FUNCTION_BLOCK FB_MotionShareData IMPLEMENTS I_MotionShareData
VAR_INPUT
END_VAR
VAR_OUTPUT
END_VAR
VAR
    (* Hardware *)
   // NC Forward Limit Switch: TRUE if ok to move
    bLimitForwardEnable AT %I*: BOOL;
    // NC Backward Limit Switch: TRUE if ok to move
    bLimitBackwardEnable AT %I*: BOOL;
    // NO Home Switch: TRUE if at home
    bHome AT %I*: BOOL;
END_VAR

{warning 'Add property implementation'}
(* Reads get this status from Interlock block*)
PROPERTY AllBackwardEnabled : BOOL
GET
END_GET
SET
END_SET
END_PROPERTY

{warning 'Add property implementation'}
(* Reads get this status from Interlock block*)
PROPERTY AllEnabled : BOOL
GET
END_GET
SET
END_SET
END_PROPERTY

{warning 'Add property implementation'}
(* Reads get this status from Interlock block*)
PROPERTY AllForwardEnabled : BOOL
GET
END_GET
SET
END_SET
END_PROPERTY

{warning 'Add property implementation'}
PROPERTY AxisError : BOOL
GET
END_GET
SET
END_SET
END_PROPERTY

{warning 'Add property implementation'}
PROPERTY AxisErrorID : UDINT
GET
END_GET
SET
END_SET
END_PROPERTY

{warning 'Add property implementation'}
PROPERTY AxisState : MC_AxisStates
GET
END_GET
SET
END_SET
END_PROPERTY

{warning 'Add property implementation'}
PROPERTY BrakeError : BOOL
GET
END_GET
END_PROPERTY

{warning 'Add property implementation'}
PROPERTY DriveEnable : BOOL
GET
END_GET
SET
END_SET
END_PROPERTY

{warning 'Add property implementation'}
PROPERTY ExecHome : BOOL
GET
END_GET
SET
END_SET
END_PROPERTY

{warning 'Add property implementation'}
PROPERTY ExecMove : BOOL
GET
END_GET
SET
END_SET
END_PROPERTY

{warning 'Add property implementation'}
PROPERTY GlobalReset : BOOL
GET
END_GET
SET
END_SET
END_PROPERTY

{warning 'Add property implementation'}
PROPERTY HomeBusy : BOOL
GET
END_GET
SET
END_SET
END_PROPERTY

{warning 'Add property implementation'}
PROPERTY InterlockOk : BOOL
GET
END_GET
END_PROPERTY

{warning 'Add property implementation'}
PROPERTY LimBackward : BOOL
GET
END_GET
END_PROPERTY

{warning 'Add property implementation'}
PROPERTY LimBwdEnable : BOOL
GET
END_GET
SET
END_SET
END_PROPERTY

{warning 'Add property implementation'}
PROPERTY LimForward : BOOL
GET
END_GET
END_PROPERTY

{warning 'Add property implementation'}
PROPERTY LimFwdEnable : BOOL
GET
END_GET
SET
END_SET
END_PROPERTY

{warning 'Add property implementation'}
PROPERTY LimHome : BOOL
GET
END_GET
SET
END_SET
END_PROPERTY

{warning 'Add property implementation'}
PROPERTY MoveBusy : BOOL
GET
END_GET
SET
END_SET
END_PROPERTY

{warning 'Add property implementation'}
PROPERTY NegativeDirection : BOOL
GET
END_GET
SET
END_SET
END_PROPERTY

{warning 'Add property implementation'}
PROPERTY NewMoveReq : BOOL
GET
END_GET
SET
END_SET
END_PROPERTY

{warning 'Add property implementation'}
PROPERTY PositiveDirection : BOOL
GET
END_GET
SET
END_SET
END_PROPERTY

{warning 'Add property implementation'}
PROPERTY ResetDone : BOOL
GET
END_GET
SET
END_SET
END_PROPERTY

{warning 'Add property implementation'}
PROPERTY RestoreDone : BOOL
GET
END_GET
SET
END_SET
END_PROPERTY

{warning 'Add property implementation'}
PROPERTY SavedPosition : LREAL
GET
END_GET
SET
END_SET
END_PROPERTY

{warning 'Add property implementation'}
PROPERTY ServoMode : BOOL
GET
END_GET
SET
END_SET
END_PROPERTY

END_FUNCTION_BLOCK

(* stored: Version 1.1.0.1
   POU FB_MotionShareData: Id {1501870c-92ad-4102-b185-4e7588eab041}, SpecialFunc None
   Property AllBackwardEnabled: Id {588933f9-668c-428c-b209-3fec4ae435c4}
   Get Get: Id {6ea50c3d-e5d3-4a80-b52c-1c3edbe55417}
   Set Set: Id {6c150d12-d1b5-4f4d-b7b7-ed56a08b0c53}
   Property AllEnabled: Id {531ae454-b142-4ec8-a6a5-51ea163f0f3b}
   Get Get: Id {35565f8a-1ea5-48a2-b92f-f1487a4c2726}
   Set Set: Id {b6605eb0-8b6e-487f-9c94-198c166233d5}
   Property AllForwardEnabled: Id {dd99efed-b46c-49c9-8796-4833ffe44a8e}
   Get Get: Id {21a84f27-171b-49b3-9d0a-8f77c1dec2a2}
   Set Set: Id {52d9b336-5323-4b37-acf3-5ca81300271c}
   Property AxisError: Id {98115272-2230-4767-b0dd-a49f097a3ce0}
   Get Get: Id {e08aea0a-ecc7-413f-a52a-c1e096c0cdf2}
   Set Set: Id {ef9e3f03-340b-499d-8070-7455ab14d8b6}
   Property AxisErrorID: Id {82dfdcd5-32b1-4e94-8a55-340757d1a7f1}
   Get Get: Id {6103d67a-1983-4236-bf4f-2f78135d229b}
   Set Set: Id {5a212e82-8ce0-4c2f-902b-ae2bc37a5cb5}
   Property AxisState: Id {cbea8871-01a0-4b37-8843-c349d6db3a77}
   Get Get: Id {b9c71475-3794-4e3a-82d7-abf6846e39f1}
   Set Set: Id {d1f98ffb-2b3d-4782-963e-39e553811b18}
   Property BrakeError: Id {b9794475-3295-45c0-b288-6d33ca0368ce}
   Get Get: Id {62ef9884-1fbf-41d5-b658-cf66ef51b265}
   Property DriveEnable: Id {dfcd0fcb-dffb-406f-b1e7-6950fa15a46c}
   Get Get: Id {db2324e9-bd6a-4fe7-9ec3-8b18495597ce}
   Set Set: Id {c3e3b36f-d36f-4e02-a404-47899aa59852}
   Property ExecHome: Id {89b20d8a-af4d-4bf3-9b64-5b77a7d8352f}
   Get Get: Id {16b7fe84-b047-4a79-80cb-896a9cb18e43}
   Set Set: Id {b29dda69-3987-4144-b0ee-0ba647ec0cf2}
   Property ExecMove: Id {91e258d6-97f4-47e1-9706-a43bc5f21419}
   Get Get: Id {a71b7848-fe39-473b-ac1e-c9df03bba908}
   Set Set: Id {3910c9d7-0829-4fb0-85f0-08cca942bd4f}
   Property GlobalReset: Id {323a9cf3-a3b0-42dc-b822-f29eb0e15c95}
   Get Get: Id {e42e6468-57d6-4eab-9213-e7eb1faa8826}
   Set Set: Id {fc8bced8-d33a-40ea-b8e4-9002dc5933ad}
   Property HomeBusy: Id {47aec562-24c8-4255-ab98-d9218f40240f}
   Get Get: Id {0cf0c789-b3ef-4e34-a21a-ea19e348b455}
   Set Set: Id {262b3e6f-6e52-4040-b215-b800b0158e51}
   Property InterlockOk: Id {3a9856fd-4650-49a0-b2fe-c96cc21117fa}
   Get Get: Id {fe0d79c1-f8f4-42e6-9406-9ec361dab8da}
   Property LimBackward: Id {38e5cd98-f346-4d1d-b128-21f2a07d0784}
   Get Get: Id {28999aa8-3674-4ecb-837f-ebb6de69864a}
   Property LimBwdEnable: Id {f6c9be89-9e8e-43ba-b22f-6910f8c266ad}
   Get Get: Id {21396ad7-f3b5-49e2-a94a-0f2ee23cefba}
   Set Set: Id {b68a63ad-3fa3-4f13-87d4-08acdd5974b5}
   Property LimForward: Id {58508ad6-a56e-4f16-90a2-2e7368217430}
   Get Get: Id {6df200ef-9186-43a2-ab57-1b46b7ba3ed7}
   Property LimFwdEnable: Id {7abd22ed-a794-45d0-86da-9a21cd25e8a9}
   Get Get: Id {ccece1fc-0a1c-4316-bb2a-391f9e29b850}
   Set Set: Id {58a697a9-c461-4dde-955a-f98b0dcfea88}
   Property LimHome: Id {4024a463-7a7f-421e-a252-cf6b7e8551bb}
   Get Get: Id {406925f6-e01e-47df-ba04-99e210a36db4}
   Set Set: Id {a7593f88-ffa7-4182-bef3-af5191879b23}
   Property MoveBusy: Id {00fdf492-934f-41b7-8610-7d81c6bd47d7}
   Get Get: Id {f877d8ca-5cdf-4313-afef-723afbba50fd}
   Set Set: Id {d1f6362a-6909-4e59-a7e3-3c32a1edb4b4}
   Property NegativeDirection: Id {36ef5103-321e-451c-b7c1-ae302c1a51ec}
   Get Get: Id {db6814e7-e4ec-451a-9d83-24d8d6e6f727}
   Set Set: Id {953a346f-5939-4424-8532-9cb60392ee2e}
   Property NewMoveReq: Id {57676e1f-cf59-4e3e-8799-1115b2803539}
   Get Get: Id {e9d5b055-8004-420d-8442-f993c0c8460b}
   Set Set: Id {61cf47b7-e6f8-4722-9380-056abd5a342b}
   Property PositiveDirection: Id {3cf963ec-fdba-444d-bdaf-38a6e7447d39}
   Get Get: Id {c80404bf-17e2-4a42-b04b-2022d416df11}
   Set Set: Id {7e41c458-a153-408d-8e1e-21815b8851e9}
   Property ResetDone: Id {7200147a-125a-4a8d-b67d-548beb5e7318}
   Get Get: Id {7a7dbf14-8bcd-452d-a365-c579db733613}
   Set Set: Id {3930e472-3ca7-4031-83ae-a2fae89bc46b}
   Property RestoreDone: Id {326c477b-e965-452d-8fa9-1f2f89e8d710}
   Get Get: Id {db53ef39-5eb5-4138-b89d-90465159112f}
   Set Set: Id {3b235ba4-2c4e-4f77-8c4e-8194d0df5e56}
   Property SavedPosition: Id {26e013d6-46e3-4463-a04e-51a04b49dcb6}
   Get Get: Id {4ac441f4-136c-439c-b9ab-415065ca001c}
   Set Set: Id {99c863ee-da0c-4b1d-918e-21040430ce54}
   Property ServoMode: Id {2a3a9bf7-5529-4d49-8d86-bcccdf694a33}
   Get Get: Id {7320238a-9fd2-47fc-b5d4-b1423e68e9ec}
   Set Set: Id {3dda8d25-c82a-4fce-9154-2ede3e832a98} *)
